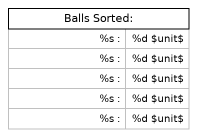
[picture p24: VC_Graph_Counters (HMI screen)]
embedded screen at (0,20)-(181,41): VC_Var_Int
rectangle at (0,0)-(181,21): text "Balls Sorted:"
embedded screen at (0,40)-(181,61): VC_Var_Int
embedded screen at (0,60)-(181,81): VC_Var_Int
embedded screen at (0,80)-(181,101): VC_Var_Int
embedded screen at (0,100)-(181,121): VC_Var_Int
*)

(* Visualisation Components/VC_GRAPH_LIFT
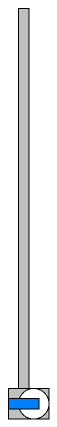
rectangle at (0,380)-(41,411): y offset -1 * PRG_HMI.iLiftPos
ellipse at (10,380)-(41,411): invisible if NOT .PRG_HMI.bBall_InLift; y offset -1 * PRG_HMI.iLiftPos
rectangle at (0,390)-(31,401): invisible if NOT .OEjector; y offset -1 * PRG_HMI.iLiftPos
1 more shapes without text or variables
*)

(* Visualisation Components/VC_GRAPH_SORTER
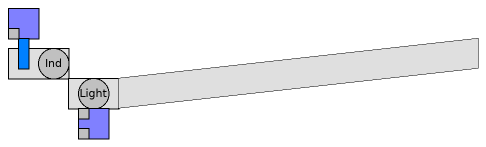
rectangle at (60,70)-(111,101): y offset -1 * PRG_HMI.iSorterLiftPos
rectangle at (10,30)-(21,61): invisible if .OSorterGate
ellipse at (70,70)-(101,101): text "Light"; alarm colour if .ISensorOpt; y offset -1 * PRG_HMI.iSorterLiftPos
ellipse at (30,40)-(61,71): text "Ind"; alarm colour if .ISensorInd
rectangle at (70,100)-(81,111): alarm colour if .ISorterLiftUp
rectangle at (70,120)-(81,131): alarm colour if .ISorterLiftDown
rectangle at (0,20)-(11,31): alarm colour if .ISorterGateClosed
6 more shapes without text or variables
*)

(* Visualisation Visual Components/VC_PackMLStates
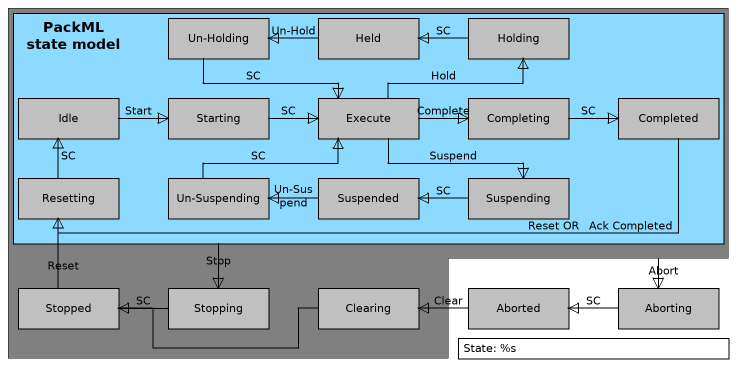
rounded rectangle at (160,280)-(261,321): text "Stopping"; alarm colour if $PackML$.eState = 4
rounded rectangle at (10,90)-(111,131): text "Idle"; alarm colour if $PackML$.eState = 6
rounded rectangle at (160,170)-(261,211): text "Un-Suspending"; alarm colour if $PackML$.eState = 11
rounded rectangle at (610,280)-(711,321): text "Aborting"; alarm colour if $PackML$.eState = 0
rounded rectangle at (460,280)-(561,321): text "Aborted"; alarm colour if $PackML$.eState = 1
rectangle at (450,330)-(721,351): text "State: %s"; shows $PackML$.strState
rounded rectangle at (310,280)-(411,321): text "Clearing"; alarm colour if $PackML$.eState = 2
rounded rectangle at (10,280)-(111,321): text "Stopped"; alarm colour if $PackML$.eState = 3
rounded rectangle at (10,170)-(111,211): text "Resetting"; alarm colour if $PackML$.eState = 5
rounded rectangle at (160,90)-(261,131): text "Starting"; alarm colour if $PackML$.eState = 7
rounded rectangle at (310,90)-(411,131): text "Execute"; alarm colour if $PackML$.eState = 8
rounded rectangle at (460,90)-(561,131): text "Completing"; alarm colour if $PackML$.eState = 15
rounded rectangle at (610,90)-(711,131): text "Completed"; alarm colour if $PackML$.eState = 16
rounded rectangle at (310,170)-(411,211): text "Suspended"; alarm colour if $PackML$.eState = 10
rounded rectangle at (460,170)-(561,211): text "Suspending"; alarm colour if $PackML$.eState = 9
rounded rectangle at (460,10)-(561,51): text "Holding"; alarm colour if $PackML$.eState = 12
rounded rectangle at (310,10)-(411,51): text "Held"; alarm colour if $PackML$.eState = 13
rounded rectangle at (160,10)-(261,51): text "Un-Holding"; alarm colour if $PackML$.eState = 14
polyline at (645,250)-(655,280): alarm colour if $PackML$.bAbort
rectangle at (635,255)-(676,271): text "Abort"; alarm colour if $PackML$.bAbort
polyline at (205,235)-(215,280): alarm colour if $PackML$.bStop
rectangle at (190,245)-(231,261): text "Stop"; alarm colour if $PackML$.bStop
polyline at (195,130)-(335,170): alarm colour if $PackML$.bSC
rectangle at (235,140)-(266,156): text "SC"; alarm colour if $PackML$.bSC
polyline at (195,50)-(335,90): alarm colour if $PackML$.bSC
polyline at (380,50)-(520,90): alarm colour if $PackML$.bHold
rectangle at (420,60)-(451,76): text "Hold"; alarm colour if $PackML$.bHold
polyline at (560,295)-(610,305): alarm colour if $PackML$.bSC
polyline at (45,210)-(55,280): alarm colour if $PackML$.bReset
polyline at (110,105)-(160,115): alarm colour if $PackML$.bStart
polyline at (110,295)-(310,340): alarm colour if $PackML$.bSC
rectangle at (230,60)-(261,76): text "SC"; alarm colour if $PackML$.bSC
polyline at (380,130)-(520,170): alarm colour if $PackML$.bSuspend
rectangle at (415,140)-(476,156): text "Suspend"; alarm colour if $PackML$.bSuspend
rectangle at (120,285)-(151,301): text "SC"; alarm colour if $PackML$.bSC
rectangle at (570,285)-(601,301): text "SC"; alarm colour if $PackML$.bSC
polyline at (410,295)-(460,305): alarm colour if $PackML$.bClear
rectangle at (420,285)-(461,301): text "Clear"; alarm colour if $PackML$.bClear
polyline at (260,105)-(310,115): alarm colour if $PackML$.bSC
rectangle at (265,95)-(296,111): text "SC"; alarm colour if $PackML$.bSC
rectangle at (110,95)-(151,111): text "Start"; alarm colour if $PackML$.bStart
rectangle at (35,250)-(76,266): text "Reset"; alarm colour if $PackML$.bReset
polyline at (410,185)-(460,195): alarm colour if $PackML$.bSC
rectangle at (420,175)-(451,191): text "SC"; alarm colour if $PackML$.bSC
polyline at (410,25)-(460,35): alarm colour if $PackML$.bSC
rectangle at (420,15)-(451,31): text "SC"; alarm colour if $PackML$.bSC
polyline at (260,185)-(310,195): alarm colour if $PackML$.bUn_Suspend
rectangle at (260,170)-(311,206): text "Un-Sus / pend"; alarm colour if $PackML$.bUn_Suspend
polyline at (260,25)-(310,35): alarm colour if $PackML$.bUn_Hold
rectangle at (260,15)-(311,31): text "Un-Hold"; alarm colour if $PackML$.bUn_Hold
polyline at (410,105)-(460,115): alarm colour if $PackML$.bComplete
rectangle at (410,95)-(461,111): text "Complete"; alarm colour if $PackML$.bComplete
polyline at (560,105)-(610,115): alarm colour if $PackML$.bSC
rectangle at (565,95)-(596,111): text "SC"; alarm colour if $PackML$.bSC
polyline at (45,130)-(55,170): alarm colour if $PackML$.bSC
rectangle at (45,140)-(76,156): text "SC"; alarm colour if $PackML$.bSC
polyline at (50,130)-(670,225): alarm colour if $PackML$.bReset OR $PackML$.Ack_Completed
rectangle at (515,210)-(576,226): text "Reset OR"; alarm colour if $PackML$.bReset
rectangle at (575,210)-(671,226): text "Ack Completed"; alarm colour if $PackML$.bAck_Completed
rectangle at (10,10)-(121,51): text "PackML / state model"
2 more shapes without text or variables
*)

(* Visualisation Simulator/MachineComponents/VC_PANEL_MACHINECONTROL
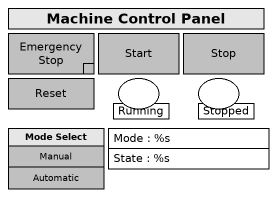
rounded rectangle at (0,25)-(86,66): text "Emergency / Stop"; alarm colour if .IEmergencyClear; toggles .IEmergencyClear
rounded rectangle at (90,25)-(171,66): text "Start"; alarm colour if .I_Btn_Start; taps .I_Btn_Start
rounded rectangle at (0,70)-(86,101): text "Reset"; alarm colour if .I_Btn_Reset; taps .I_Btn_Reset
rounded rectangle at (175,25)-(256,66): text "Stop"; alarm colour if .I_Btn_Stop; taps .I_Btn_Stop
rectangle at (0,0)-(256,21): text "Machine Control Panel"
rectangle at (100,120)-(261,141): text "Mode : %s"; shows .fbStateModel.eMode
rectangle at (100,140)-(261,161): text "State : %s"; shows .fbStateModel.eState
embedded screen at (0,120)-(96,181): VC_Panel_ModeSelector
rectangle at (105,95)-(161,111): text "Running"
rectangle at (190,95)-(246,111): text "Stopped"
ellipse at (110,70)-(151,101): alarm colour if .O_Light_Start
ellipse at (190,70)-(231,101): alarm colour if .O_Light_Stop
embedded screen at (75,55)-(86,66): VC_sensor
*)

(* Visualisation Simulator/MachineComponents/VC_PANEL_MODESELECTOR
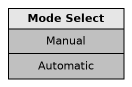
rounded rectangle at (0,20)-(116,46): text "Manual"; alarm colour if .HMI_uModeReq=3; runs INTERN ASSIGN HMI_uModeReq:=(3)
rectangle at (0,0)-(116,21): text "Mode Select"
rounded rectangle at (0,45)-(116,71): text "Automatic"; alarm colour if .HMI_uModeReq=1; runs INTERN ASSIGN HMI_uModeReq:=(1)
*)

(* Visualisation Simulator/Components/VC_sensor
rectangle at (0,0)-(11,11): alarm colour if $VAR$
*)

(* Visualisation Components/VC_Var_Int
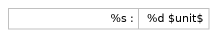
rectangle at (0,0)-(131,21): text "%s :"; shows $Name$
rectangle at (130,0)-(201,21): text "%d $unit$"; shows $VAR$
*)
